// TIA Portal V20 export
DATA_BLOCK "Data"   // DB40
// stored: Access Published, MemoryReserve 100, Namespace Global
   VAR
      general : "LAF_typeGeneralStatus";   // Global status information
      unit : Array[0.._.NO_OF_UNITS] of "LAF_typeUnitInterface";   // Global information of units
   END_VAR
BEGIN
   general.acknowledge := FALSE;
   general.disableAlarms := FALSE;
   general.activateSimulation := TRUE;
   general.enablePower := FALSE;   // Power is off. Switch on!
   general.localPlcDateAndTime.retVal := 0;
   general.localPlcDateAndTime.dtl := DTL#2026-01-06-19:57:49.792575863;
   general.localPlcDateAndTime.ldt := LDT#2026-01-06-19:57:49.792575863;
   general.localPlcDateAndTime."dt" := DT#2026-01-06-19:57:49.792;
   general.dayLightSavingTime := FALSE;
   general.clock.cycle100Msec := TRUE;
   general.clock.cycle200Msec := TRUE;
   general.clock.cycle400Msec := TRUE;
   general.clock.cycle500Msec := FALSE;
   general.clock.cycle800Msec := FALSE;
   general.clock.cycle1000Msec := FALSE;
   general.clock.cycle1600Msec := TRUE;
   general.clock.cycle2000Msec := TRUE;
   general.posPulse.cycle100Msec := FALSE;
   general.posPulse.cycle200Msec := FALSE;
   general.posPulse.cycle400Msec := FALSE;
   general.posPulse.cycle500Msec := FALSE;
   general.posPulse.cycle800Msec := FALSE;
   general.posPulse.cycle1000Msec := FALSE;
   general.posPulse.cycle1600Msec := FALSE;
   general.posPulse.cycle2000Msec := FALSE;
   general.clockMemoryByte := 16#C7;
   general.firstCycle := FALSE;
   unit[0].information.equipmentID := 0;
   unit[0].information.equipmentName := WSTRING#'';
   unit[0].information.equipmentVersion := WSTRING#'';
   unit[0].information.interfaceVersionProject := WSTRING#'';
   unit[0].information.lineID := 0;
   unit[0].information.vendorID := 0;
   unit[0].status.designSpeed := 0.0;
   unit[0].status.currentSpeed := 0.0;
   unit[0].status.totalCounter := 0;
   unit[0].status.goodCounter := 0;
   unit[0].enableControlInterfaces.local := TRUE;
   unit[0].enableControlInterfaces.hmi := FALSE;
   unit[0].enableControlInterfaces.remote := FALSE;
   unit[0].controlModeStateManager.commands.modeRequests.production := FALSE;
   unit[0].controlModeStateManager.commands.modeRequests.maintenance := FALSE;
   unit[0].controlModeStateManager.commands.modeRequests.manual := FALSE;
   unit[0].controlModeStateManager.commands.modeRequests.nomode := FALSE;
   unit[0].controlModeStateManager.commands.modeRequests.sleep := FALSE;
   unit[0].controlModeStateManager.commands.modeRequests.deepsleep := FALSE;
   unit[0].controlModeStateManager.commands.modeRequests.userMode04 := FALSE;
   unit[0].controlModeStateManager.commands.modeRequests.userMode05 := FALSE;
   unit[0].controlModeStateManager.commands.modeRequests.userMode06 := FALSE;
   unit[0].controlModeStateManager.commands.modeRequests.userMode07 := FALSE;
   unit[0].controlModeStateManager.commands.modeRequests.userMode08 := FALSE;
   unit[0].controlModeStateManager.commands.modeRequests.userMode09 := FALSE;
   unit[0].controlModeStateManager.commands.modeRequests.userMode10 := FALSE;
   unit[0].controlModeStateManager.commands.modeRequests.userMode11 := FALSE;
   unit[0].controlModeStateManager.commands.modeRequests.userMode12 := FALSE;
   unit[0].controlModeStateManager.commands.modeRequests.userMode13 := FALSE;
   unit[0].controlModeStateManager.commands.stateCommands.reset := FALSE;
   unit[0].controlModeStateManager.commands.stateCommands.start := FALSE;
   unit[0].controlModeStateManager.commands.stateCommands.stop := FALSE;
   unit[0].controlModeStateManager.commands.stateCommands.hold := FALSE;
   unit[0].controlModeStateManager.commands.stateCommands.unhold := FALSE;
   unit[0].controlModeStateManager.commands.stateCommands.suspend := FALSE;
   unit[0].controlModeStateManager.commands.stateCommands.unsuspend := FALSE;
   unit[0].controlModeStateManager.commands.stateCommands.abort := FALSE;
   unit[0].controlModeStateManager.commands.stateCommands.clear := FALSE;
   unit[0].controlModeStateManager.commands.stateCommands.complete := FALSE;
   unit[0].controlModeStateManager.commands.stateCommands.stateComplete := FALSE;
   unit[0].controlModeStateManager.monitoring.unitModeCurrent := 2;
   unit[0].controlModeStateManager.monitoring.unitModeRequested := FALSE;
   unit[0].controlModeStateManager.monitoring.unitModeChangeInProcess := FALSE;
   unit[0].controlModeStateManager.monitoring.stateCurrent := 2;
   unit[0].controlModeStateManager.monitoring.stateRequested := 2;
   unit[0].controlModeStateManager.monitoring.stateChangeInProcess := FALSE;
   unit[0].controlModeStateManager.monitoring.curDisabledStates := 16#0003_6020;
   unit[0].controlModeStateManager.monitoring.curHoldCmdCfg := 16#0000_0040;
   unit[0].controlModeStateManager.monitoring.curCompleteCmdCfg := 16#0000_0000;
   unit[0].controlModeStateManager.monitoring.curEnabledModes := 16#0000_007F;
   unit[0].controlModeStateManager.monitoring.allowedUnitModes := 16#0000_001A;
   unit[0].controlModeStateManager.monitoring.cntrlCmdNotAllowed := FALSE;
   unit[0].controlModeStateManager.monitoring.localControlEnabled := TRUE;
   unit[0].controlModeStateManager.monitoring.hmiControlEnabled := FALSE;
   unit[0].controlModeStateManager.monitoring.remoteControlEnabled := FALSE;
   unit[0].controlModeStateManager.diagnostics.interfaceManagerStatus := 16#0000;
   unit[0].controlModeStateManager.diagnostics.modeStateManagerDiagnostics.bufferIndex := 7;
   unit[0].controlModeStateManager.diagnostics.modeStateManagerDiagnostics.buffer[0].timestamp := DTL#2026-01-06-06:46:51.371465172;
   unit[0].controlModeStateManager.diagnostics.modeStateManagerDiagnostics.buffer[1].timestamp := DTL#2026-01-06-06:46:51.374585015;
   unit[0].controlModeStateManager.diagnostics.modeStateManagerDiagnostics.buffer[2].timestamp := DTL#2026-01-06-06:46:51.567016868;
   unit[0].controlModeStateManager.diagnostics.modeStateManagerDiagnostics.buffer[3].timestamp := DTL#2026-01-06-06:46:55.878705971;
   unit[0].controlModeStateManager.diagnostics.modeStateManagerDiagnostics.buffer[4].timestamp := DTL#2026-01-06-06:46:55.971592245;
   unit[0].controlModeStateManager.diagnostics.modeStateManagerDiagnostics.buffer[5].timestamp := DTL#2026-01-06-06:46:58.882031211;
   unit[0].controlModeStateManager.diagnostics.modeStateManagerDiagnostics.buffer[6].timestamp := DTL#2026-01-06-06:46:58.884831167;
   unit[0].controlModeStateManager.diagnostics.modeStateManagerDiagnostics.buffer[7].timestamp := DTL#2026-01-06-06:46:58.887783077;
   unit[0].controlModeStateManager.diagnostics.modeStateManagerDiagnostics.buffer[0..2].UnitModeCurrent := 2;
   unit[0].controlModeStateManager.diagnostics.modeStateManagerDiagnostics.buffer[3..6].UnitModeCurrent := 4;
   unit[0].controlModeStateManager.diagnostics.modeStateManagerDiagnostics.buffer[7].UnitModeCurrent := 2;
   unit[0].controlModeStateManager.diagnostics.modeStateManagerDiagnostics.buffer[0].StateCurrent := 8;
   unit[0].controlModeStateManager.diagnostics.modeStateManagerDiagnostics.buffer[1..3].StateCurrent := 9;
   unit[0].controlModeStateManager.diagnostics.modeStateManagerDiagnostics.buffer[4..5].StateCurrent := 1;
   unit[0].controlModeStateManager.diagnostics.modeStateManagerDiagnostics.buffer[6..7].StateCurrent := 2;
   unit[0].controlModeStateManager.diagnostics.modeStateManagerDiagnostics.buffer[0].UnitMode := 0;
   unit[0].controlModeStateManager.diagnostics.modeStateManagerDiagnostics.buffer[1].UnitMode := 2;
   unit[0].controlModeStateManager.diagnostics.modeStateManagerDiagnostics.buffer[2].UnitMode := 4;
   unit[0].controlModeStateManager.diagnostics.modeStateManagerDiagnostics.buffer[3..5].UnitMode := 0;
   unit[0].controlModeStateManager.diagnostics.modeStateManagerDiagnostics.buffer[6].UnitMode := 2;
   unit[0].controlModeStateManager.diagnostics.modeStateManagerDiagnostics.buffer[7].UnitMode := 0;
   unit[0].controlModeStateManager.diagnostics.modeStateManagerDiagnostics.buffer[0..2].CntrlCmd := 8;
   unit[0].controlModeStateManager.diagnostics.modeStateManagerDiagnostics.buffer[3].CntrlCmd := 9;
   unit[0].controlModeStateManager.diagnostics.modeStateManagerDiagnostics.buffer[4..7].CntrlCmd := 3;
   unit[0].controlModeStateManager.diagnostics.modeStateManagerDiagnostics.buffer[0].SC := TRUE;
   unit[0].controlModeStateManager.diagnostics.modeStateManagerDiagnostics.buffer[1..4].SC := FALSE;
   unit[0].controlModeStateManager.diagnostics.modeStateManagerDiagnostics.buffer[5].SC := TRUE;
   unit[0].controlModeStateManager.diagnostics.modeStateManagerDiagnostics.buffer[6].SC := FALSE;
   unit[0].controlModeStateManager.diagnostics.modeStateManagerDiagnostics.buffer[7].SC := TRUE;
   unit[0].controlModeStateManager.diagnostics.modeStateManagerDiagnostics.buffer[0].message := 16#02;
   unit[0].controlModeStateManager.diagnostics.modeStateManagerDiagnostics.buffer[1].message := 16#03;
   unit[0].controlModeStateManager.diagnostics.modeStateManagerDiagnostics.buffer[2].message := 16#01;
   unit[0].controlModeStateManager.diagnostics.modeStateManagerDiagnostics.buffer[3].message := 16#02;
   unit[0].controlModeStateManager.diagnostics.modeStateManagerDiagnostics.buffer[4].message := 16#84;
   unit[0].controlModeStateManager.diagnostics.modeStateManagerDiagnostics.buffer[5].message := 16#02;
   unit[0].controlModeStateManager.diagnostics.modeStateManagerDiagnostics.buffer[6].message := 16#01;
   unit[0].controlModeStateManager.diagnostics.modeStateManagerDiagnostics.buffer[7].message := 16#85;
   unit[0].signalStack.statusByDWord := 16#0000_0000;
   unit[0].currentMode := 'Maintenance';
   unit[0].currentState := 'Stopped';
   unit[0].history[0].mode := 2;
   unit[0].history[1..3].mode := 4;
   unit[0].history[4..6].mode := 2;
   unit[0].history[7..9].mode := 4;
   unit[0].history[10].mode := 2;
   unit[0].history[11..14].mode := 4;
   unit[0].history[15].mode := 2;
   unit[0].history[0..1].state := 2;
   unit[0].history[2].state := 1;
   unit[0].history[3..4].state := 9;
   unit[0].history[5].state := 8;
   unit[0].history[6..7].state := 2;
   unit[0].history[8].state := 1;
   unit[0].history[9..11].state := 9;
   unit[0].history[12].state := 8;
   unit[0].history[13].state := 1;
   unit[0].history[14..15].state := 9;
   unit[0].history[0].duration := 2.7196749144815E-308;
   unit[0].history[1].duration := 0.00280152420343137;
   unit[0].history[2].duration := 3.00332605851716;
   unit[0].history[3].duration := 4.31168274203431;
   unit[0].history[4].duration := 0.195557047334559;
   unit[0].history[5].duration := 0.00613084712009804;
   unit[0].history[6].duration := 14200.181291368;
   unit[0].history[7].duration := 0.00276850566789216;
   unit[0].history[8].duration := 3.00295925245098;
   unit[0].history[9].duration := 0.812557797947304;
   unit[0].history[10].duration := 0.0728598659620098;
   unit[0].history[11].duration := 0.00270324754901961;
   unit[0].history[12].duration := 0.00544693857230392;
   unit[0].history[13].duration := 2.00414811810662;
   unit[0].history[14].duration := 1.31479962775735;
   unit[0].history[15].duration := 0.194273973651961;
   unit[0].modeStateTimeStatistics.modeTimeCurrent := 47450;
   unit[0].modeStateTimeStatistics.stateTimeCurrent := 47450;
   unit[0].modeStateTimeStatistics.accTimeSinceReset := 71286;
   unit[0].modeStateTimeStatistics.actualTimeAllModes[0..1] := 0;
   unit[0].modeStateTimeStatistics.actualTimeAllModes[2] := 47450;
   unit[0].modeStateTimeStatistics.actualTimeAllModes[3] := 0;
   unit[0].modeStateTimeStatistics.actualTimeAllModes[4] := 8;
   unit[0].modeStateTimeStatistics.actualTimeAllModes[5..16] := 0;
   unit[0].modeStateTimeStatistics.cumulativeTimeAllModes[0..1] := 0;
   unit[0].modeStateTimeStatistics.cumulativeTimeAllModes[2] := 67850;
   unit[0].modeStateTimeStatistics.cumulativeTimeAllModes[3] := 0;
   unit[0].modeStateTimeStatistics.cumulativeTimeAllModes[4] := 3436;
   unit[0].modeStateTimeStatistics.cumulativeTimeAllModes[5..16] := 0;
   unit[0].modeStateTimeStatistics.actualTimeAllStatesOfAllModes[0,0..17] := 0;
   unit[0].modeStateTimeStatistics.actualTimeAllStatesOfAllModes[1,0..17] := 0;
   unit[0].modeStateTimeStatistics.actualTimeAllStatesOfAllModes[2,0] := 0;
   unit[0].modeStateTimeStatistics.actualTimeAllStatesOfAllModes[2,1] := 3;
   unit[0].modeStateTimeStatistics.actualTimeAllStatesOfAllModes[2,2] := 47450;
   unit[0].modeStateTimeStatistics.actualTimeAllStatesOfAllModes[2,3..17] := 0;
   unit[0].modeStateTimeStatistics.actualTimeAllStatesOfAllModes[3,0..17] := 0;
   unit[0].modeStateTimeStatistics.actualTimeAllStatesOfAllModes[4,0] := 0;
   unit[0].modeStateTimeStatistics.actualTimeAllStatesOfAllModes[4,1] := 3;
   unit[0].modeStateTimeStatistics.actualTimeAllStatesOfAllModes[4,2..8] := 0;
   unit[0].modeStateTimeStatistics.actualTimeAllStatesOfAllModes[4,9] := 5;
   unit[0].modeStateTimeStatistics.actualTimeAllStatesOfAllModes[4,10..17] := 0;
   unit[0].modeStateTimeStatistics.actualTimeAllStatesOfAllModes[5,0..17] := 0;
   unit[0].modeStateTimeStatistics.actualTimeAllStatesOfAllModes[6,0..17] := 0;
   unit[0].modeStateTimeStatistics.actualTimeAllStatesOfAllModes[7,0..17] := 0;
   unit[0].modeStateTimeStatistics.actualTimeAllStatesOfAllModes[8,0..17] := 0;
   unit[0].modeStateTimeStatistics.actualTimeAllStatesOfAllModes[9,0..17] := 0;
   unit[0].modeStateTimeStatistics.actualTimeAllStatesOfAllModes[10,0..17] := 0;
   unit[0].modeStateTimeStatistics.actualTimeAllStatesOfAllModes[11,0..17] := 0;
   unit[0].modeStateTimeStatistics.actualTimeAllStatesOfAllModes[12,0..17] := 0;
   unit[0].modeStateTimeStatistics.actualTimeAllStatesOfAllModes[13,0..17] := 0;
   unit[0].modeStateTimeStatistics.actualTimeAllStatesOfAllModes[14,0..17] := 0;
   unit[0].modeStateTimeStatistics.actualTimeAllStatesOfAllModes[15,0..17] := 0;
   unit[0].modeStateTimeStatistics.actualTimeAllStatesOfAllModes[16,0..17] := 0;
   unit[0].modeStateTimeStatistics.cumulativeTimeAllStatesOfAllModes[0,0..17] := 0;
   unit[0].modeStateTimeStatistics.cumulativeTimeAllStatesOfAllModes[1,0..17] := 0;
   unit[0].modeStateTimeStatistics.cumulativeTimeAllStatesOfAllModes[2,0] := 0;
   unit[0].modeStateTimeStatistics.cumulativeTimeAllStatesOfAllModes[2,1] := 29;
   unit[0].modeStateTimeStatistics.cumulativeTimeAllStatesOfAllModes[2,2] := 62969;
   unit[0].modeStateTimeStatistics.cumulativeTimeAllStatesOfAllModes[2,3..7] := 0;
   unit[0].modeStateTimeStatistics.cumulativeTimeAllStatesOfAllModes[2,8] := 1;
   unit[0].modeStateTimeStatistics.cumulativeTimeAllStatesOfAllModes[2,9] := 4851;
   unit[0].modeStateTimeStatistics.cumulativeTimeAllStatesOfAllModes[2,10..17] := 0;
   unit[0].modeStateTimeStatistics.cumulativeTimeAllStatesOfAllModes[3,0..17] := 0;
   unit[0].modeStateTimeStatistics.cumulativeTimeAllStatesOfAllModes[4,0] := 0;
   unit[0].modeStateTimeStatistics.cumulativeTimeAllStatesOfAllModes[4,1] := 35;
   unit[0].modeStateTimeStatistics.cumulativeTimeAllStatesOfAllModes[4,2..8] := 0;
   unit[0].modeStateTimeStatistics.cumulativeTimeAllStatesOfAllModes[4,9] := 3401;
   unit[0].modeStateTimeStatistics.cumulativeTimeAllStatesOfAllModes[4,10..17] := 0;
   unit[0].modeStateTimeStatistics.cumulativeTimeAllStatesOfAllModes[5,0..17] := 0;
   unit[0].modeStateTimeStatistics.cumulativeTimeAllStatesOfAllModes[6,0..17] := 0;
   unit[0].modeStateTimeStatistics.cumulativeTimeAllStatesOfAllModes[7,0..17] := 0;
   unit[0].modeStateTimeStatistics.cumulativeTimeAllStatesOfAllModes[8,0..17] := 0;
   unit[0].modeStateTimeStatistics.cumulativeTimeAllStatesOfAllModes[9,0..17] := 0;
   unit[0].modeStateTimeStatistics.cumulativeTimeAllStatesOfAllModes[10,0..17] := 0;
   unit[0].modeStateTimeStatistics.cumulativeTimeAllStatesOfAllModes[11,0..17] := 0;
   unit[0].modeStateTimeStatistics.cumulativeTimeAllStatesOfAllModes[12,0..17] := 0;
   unit[0].modeStateTimeStatistics.cumulativeTimeAllStatesOfAllModes[13,0..17] := 0;
   unit[0].modeStateTimeStatistics.cumulativeTimeAllStatesOfAllModes[14,0..17] := 0;
   unit[0].modeStateTimeStatistics.cumulativeTimeAllStatesOfAllModes[15,0..17] := 0;
   unit[0].modeStateTimeStatistics.cumulativeTimeAllStatesOfAllModes[16,0..17] := 0;
   unit[0].modeStateTimeStatistics.actualTimeAllStatesOfCurrentMode[0] := 0;
   unit[0].modeStateTimeStatistics.actualTimeAllStatesOfCurrentMode[1] := 3;
   unit[0].modeStateTimeStatistics.actualTimeAllStatesOfCurrentMode[2] := 47450;
   unit[0].modeStateTimeStatistics.actualTimeAllStatesOfCurrentMode[3..17] := 0;
   unit[0].modeStateTimeStatistics.cumulativeTimeAllStatesOfCurrentMode[0] := 0;
   unit[0].modeStateTimeStatistics.cumulativeTimeAllStatesOfCurrentMode[1] := 29;
   unit[0].modeStateTimeStatistics.cumulativeTimeAllStatesOfCurrentMode[2] := 62969;
   unit[0].modeStateTimeStatistics.cumulativeTimeAllStatesOfCurrentMode[3..7] := 0;
   unit[0].modeStateTimeStatistics.cumulativeTimeAllStatesOfCurrentMode[8] := 1;
   unit[0].modeStateTimeStatistics.cumulativeTimeAllStatesOfCurrentMode[9] := 4851;
   unit[0].modeStateTimeStatistics.cumulativeTimeAllStatesOfCurrentMode[10..17] := 0;
   unit[0].modeStateTimeStatistics.cumulativeTimeCurrentMode := 67850;
END_DATA_BLOCK
